FUNCTION_BLOCK InsertionSequence
VAR_IN_OUT
	
END_VAR
VAR
	insertion : PneumaticInsertion;
	
	contUp, contDown : BOOL;
	vTarget : REAL := -1;
	press, release : BOOL;
END_VAR

insertion(
	enable:= TRUE, 
	slider=> , 
	screw=> , 
	contact=> , 
	home=> , 
	ready=> , 
	busy=> , 
	error=> , 
	homeSet=> );

IF NOT insertion.homeSet THEN
	insertion.homingSequence();
	RETURN;
END_IF

insertion.stop(); //executes if any of the following are false

IF contUp THEN
	insertion.slideContinuous(direction := MC_Positive_Direction);
	contDown := FALSE;
END_IF

IF contDown THEN
	insertion.slideContinuous(direction := MC_Negative_Direction);
	contUp := FALSE;
END_IF

IF vTarget >= 0 THEN
	insertion.slideAbsolute(targetPos := vTarget);
END_IF

END_FUNCTION_BLOCK

(* stored: Version 1.1.0.1, ProductVersion 3.1.4024.11
   POU InsertionSequence: Id {4c77553f-a0fc-426c-82d7-73e96ddccd49}, SpecialFunc None *)
